FUNCTION_BLOCK InfluentFeedLogic (* CAT Function Block Type *)
  (* Standard: 61499-2 *)
  (* Version 0.0, 6/13/2026, Schneider Electric, template *)
  PACKAGE SE.Nereda;
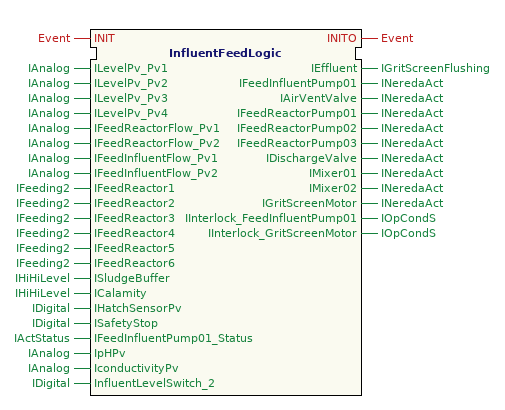
  EVENT_INPUT
    INIT;
  END_EVENT
  EVENT_OUTPUT
    INITO;
  END_EVENT
  SOCKETS
    ILevelPv_Pv1 : IAnalog;
    ILevelPv_Pv2 : IAnalog;
    ILevelPv_Pv3 : IAnalog;
    ILevelPv_Pv4 : IAnalog;
    IFeedReactorFlow_Pv1 : IAnalog;
    IFeedReactorFlow_Pv2 : IAnalog;
    IFeedInfluentFlow_Pv1 : IAnalog;
    IFeedInfluentFlow_Pv2 : IAnalog; (* Process value (range considered) interface adapter *)
    IFeedReactor1 : IFeeding2;
    IFeedReactor2 : IFeeding2;
    IFeedReactor3 : IFeeding2;
    IFeedReactor4 : IFeeding2;
    IFeedReactor5 : IFeeding2;
    IFeedReactor6 : IFeeding2;
    ISludgeBuffer : IHiHiLevel;
    ICalamity : IHiHiLevel;
    IHatchSensorPv : IDigital;
    ISafetyStop : IDigital;
    IFeedInfluentPump01_Status : IActStatus;
    IpHPv : IAnalog;
    IconductivityPv : IAnalog;
    InfluentLevelSwitch_2 : IDigital;
  END_SOCKETS
  PLUGS
    IEffluent : IGritScreenFlushing;
  END_PLUGS
  PLUGS
    IFeedInfluentPump01 : INeredaAct;
    IAirVentValve : INeredaAct;
    IFeedReactorPump01 : INeredaAct;
    IFeedReactorPump02 : INeredaAct;
    IFeedReactorPump03 : INeredaAct;
    IDischargeValve : INeredaAct;
    IMixer01 : INeredaAct;
    IMixer02 : INeredaAct;
    IGritScreenMotor : INeredaAct;
    IInterlock_FeedInfluentPump01 : IOpCondS; (* Condition summary chain output to downstream block *)
    IInterlock_GritScreenMotor : IOpCondS; (* Condition summary chain output to downstream block *)
  END_PLUGS
  (* 01 - FUNCTIONNAL INPUT INTERFACE *)
  (* 00 - INITIALIZATION *)
  (* 05 - LOGIC *)
  (* 06 - HMI INTERFACE *)
  (* 03 - FIELD INTERFACE *)
  (* Feed -> InfluentFeed   (Pump : 46 2 AP ifp 95 001) *)
  (* 02 - FUNCTIONNAL OUTPUT INTERFACE *)
  (* InfluentFeed -> Drain   (Pump : NVPP 001 ctp 001) *)
  (* Grit Screen Logic   (Motor : NVPP 001 RGI 001) *)
  (* Mixer Logic   (Motor : NVPP 001 mng 001) *)
  FBS
    Feed_InfluentFeed : FeedInfluentLogic;
    Drain_InfluentFeed : FeedReactorLogic;
    GritScreenLogic : GritScreenLogic;
    Mixer01Logic : MixerLogic;
    IThis : InfluentFeedLogic_HMI(QI := TRUE);
    Mixer02Logic : MixerLogic;
  END_FBS
  EVENT_CONNECTIONS
    INIT TO IThis.2E8F877B586EB741;
    IThis.E6EF5A4388927AD8 TO Feed_InfluentFeed.58FEB60020BBACE1;
    Feed_InfluentFeed.3BFFB52EC3F9CDAC TO Drain_InfluentFeed.58FEB60020BBACE1;
    IEffluent.0804B8CDC1B712F8 TO Feed_InfluentFeed.E90355DA9919CF7F;
    IEffluent.727D767C86127C4D TO Feed_InfluentFeed.3E2D5FB96282659D;
    Feed_InfluentFeed.E12A546BA34B0743 TO IEffluent.469E3B76B9D721DD;
    Feed_InfluentFeed.442D9E39AAC2E640 TO IEffluent.9EB419218931A109;
    Drain_InfluentFeed.3BFFB52EC3F9CDAC TO GritScreenLogic.0996BAD8F769B915;
    Drain_InfluentFeed.83AE2D5C5FB1EDB1 TO IEffluent.1F1020E82AE58441;
    IEffluent.9850048ED095E451 TO GritScreenLogic.ADE4DE4A76538746;
    GritScreenLogic.1EA29378D87A8B35 TO Mixer01Logic.66FB3AFD4368DC76;
    GritScreenLogic.3A6B5E8C5702FBA3 TO IEffluent.8B235293E5389BC7;
    Mixer02Logic.2BF2F6D7B5DAD30F TO INITO;
    Drain_InfluentFeed.444B7C715B0CFEB8 TO IEffluent.84E5BD043B0B9D2B;
    Mixer01Logic.2BF2F6D7B5DAD30F TO Mixer02Logic.66FB3AFD4368DC76;
  END_CONNECTIONS
  DATA_CONNECTIONS
    IEffluent.F5105E8545B1ACE0 TO Feed_InfluentFeed.8F3537DDF29E82C2;
    IEffluent.3A1846690B174C3E TO Feed_InfluentFeed.FC2B1174FF2CA02F;
    Feed_InfluentFeed.06D7D27D6B83410B TO IEffluent.DB5751043930F3B0;
    Feed_InfluentFeed.FA6EA9D5065FD640 TO IEffluent.76B4FEAFDB90B7B7;
    Feed_InfluentFeed.4556A9C1C2CFEDA9 TO IEffluent.B8A74FB92C78BAA2;
    Drain_InfluentFeed.6AA41E05F8773D91 TO IEffluent.E2165610E67441AB;
    Drain_InfluentFeed.1EDBE6D715573534 TO IEffluent.48F01954AB34CBCD;
    IEffluent.9EB3C16A25E3E4D9 TO GritScreenLogic.76D0FEE710977B1E;
    GritScreenLogic.CA5517AE7339BA90 TO IEffluent.CA59F9F3463F604B;
    GritScreenLogic.16751299E2E45838 TO IEffluent.917420DCD3928957;
    Drain_InfluentFeed.9351EF04351FE70A TO IEffluent.1B5136012ECA25B4;
  END_CONNECTIONS
  ADAPTER_CONNECTIONS
    ILevelPv_Pv1 TO Feed_InfluentFeed.2B8BA8A9171D2175;
    IFeedInfluentFlow_Pv1 TO Feed_InfluentFeed.91BC9C478E4F810A;
    ISludgeBuffer TO Feed_InfluentFeed.348D5C81E951271C;
    ICalamity TO Feed_InfluentFeed.BC8591F314A1A575;
    IFeedInfluentFlow_Pv2 TO Feed_InfluentFeed.2C367CE2AE2DAA6C;
    Feed_InfluentFeed.2C8DFF133A7800EF TO IFeedInfluentPump01;
    Feed_InfluentFeed.F8EDB194F3D98DD8 TO Drain_InfluentFeed.78F509CE353EF376;
    Feed_InfluentFeed.B3808BAF5CF56D5D TO IInterlock_FeedInfluentPump01;
    ILevelPv_Pv2 TO Drain_InfluentFeed.2B8BA8A9171D2175;
    IFeedReactorFlow_Pv1 TO Drain_InfluentFeed.91BC9C478E4F810A;
    IFeedReactor1 TO Drain_InfluentFeed.B12D6BA38D52F15D;
    IFeedReactor2 TO Drain_InfluentFeed.02CA94B1D7D3AA0C;
    IFeedReactor3 TO Drain_InfluentFeed.9B88906739AEC777;
    IFeedReactor4 TO Drain_InfluentFeed.B532FDFB8EF1C91A;
    IFeedReactor5 TO Drain_InfluentFeed.C88CF5C288C3B37B;
    IFeedReactor6 TO Drain_InfluentFeed.5660831129E248EB;
    IFeedReactorFlow_Pv2 TO Drain_InfluentFeed.2C367CE2AE2DAA6C;
    Drain_InfluentFeed.2C8DFF133A7800EF TO IFeedReactorPump01;
    Drain_InfluentFeed.070BC8C59167FAF7 TO IDischargeValve;
    IHatchSensorPv TO GritScreenLogic.52077DCC61F0B1BD;
    ISafetyStop TO GritScreenLogic.F4DF5A3184FB932D;
    IFeedInfluentPump01_Status TO GritScreenLogic.93E8B22DB41CD544;
    GritScreenLogic.BFB03C5769C7401A TO IGritScreenMotor;
    ILevelPv_Pv3 TO Mixer01Logic.9EEED033168D712F;
    Mixer01Logic.B800EAF158E6D272 TO IMixer01;
    Feed_InfluentFeed.9B8B0554FED936E6 TO IAirVentValve;
    GritScreenLogic.04485FF8C96F2743 TO IInterlock_GritScreenMotor;
    ILevelPv_Pv4 TO Mixer02Logic.9EEED033168D712F;
    Mixer02Logic.B800EAF158E6D272 TO IMixer02;
    Drain_InfluentFeed.2249F314E83A5F29 TO IFeedReactorPump02;
    Drain_InfluentFeed.A1E3E5AFDC140E6A TO IFeedReactorPump03;
    IpHPv TO Drain_InfluentFeed.81AEF12EA56507EE;
    IconductivityPv TO Drain_InfluentFeed.3B148542855EADBC;
    InfluentLevelSwitch_2 TO Drain_InfluentFeed.D839FD16A23DBF75;
  END_CONNECTIONS
END_FUNCTION_BLOCK
